// TwinCAT 3 PLC project TimeLogger_Plc
// ProgramVersion: 3.1.4023.0
// libraries:
//   Tc2_Standard, * (Beckhoff Automation GmbH)
//   Tc2_System, * (Beckhoff Automation GmbH)
//   Tc2_Utilities, * (Beckhoff Automation GmbH)
//   Tc3_Module, * (Beckhoff Automation GmbH)
// project tree:
//   DUTs/ E_EventType.TcDUT, ST_Event.TcDUT
//   / PlcTask.TcTTO
//   POUs/ EventLogger.TcPOU, FB_CsvPersistentEventStorage.TcPOU, I_PersistentEventStorage.TcIO, MAIN.TcPOU, UpdateEventTimestampWithSystemTime.TcPOU

CONFIGURATION TimeLogger_Plc
    RESOURCE PLC ON TwinCAT3
        TASK PlcTask(INTERVAL := T#10ms, PRIORITY := 20);
        PROGRAM MAIN WITH PlcTask : MAIN;
    END_RESOURCE
END_CONFIGURATION

// ---- DUTs/E_EventType.TcDUT
{attribute 'qualified_only'}
{attribute 'strict'}
{attribute 'to_string'}
TYPE E_EventType :
(
	Alarm := 0,
	Message := 1
);
END_TYPE

// ---- DUTs/ST_Event.TcDUT
TYPE ST_Event :
STRUCT
	eEventType : E_EventType; //user defined ENUM
	eEventSeverity : TcEventSeverity; // library ENUM
	nEventIdentity : UDINT;
	sEvenText : STRING(255);
	dtTimestamp : DATE_AND_TIME;
END_STRUCT
END_TYPE

// ---- POUs/I_PersistentEventStorage.TcIO
INTERFACE I_PersistentEventStorage

METHOD StoreEvent
VAR_INPUT
	stEvent : ST_Event;
END_VAR
END_METHOD

END_INTERFACE

// ---- POUs/MAIN.TcPOU
PROGRAM MAIN
VAR
	// Boolean to execute the Eventlogger in one PLC cycle
	bBoolean : BOOL := FALSE; 
	
	// Define sample values to the variables needed to add an Event
	eEventType1 : E_EventType := E_EventType.Alarm; //user defined ENUM
	eEventSeverity1 : TcEventSeverity := TcEventSeverity.Error; // library ENUM
	nEventIdentity1 : UDINT := 42;
	sEvenText1 : STRING(255) := 'This is a sample event';
	
	// Create an instance of the FB that defines the format for Persistent Event Storage
	CsvPersistentEventStorage1 : FB_CsvPersistentEventStorage;
	
	// Create one instance of our FB EventLogger, and provide interface parameter for FB_init
	EventLogger1 : EventLogger(CsvPersistentEventStorage1); 
	
END_VAR

IF bBoolean THEN
	// Add an event (in one cycle of the PLC)
	EventLogger1.AddEvent(eEventType1, eEventSeverity1, nEventIdentity1, sEvenText1); 
	bBoolean := FALSE;
END_IF

// call instance every cycle
CsvPersistentEventStorage1();

END_PROGRAM

// ---- POUs/FB_CsvPersistentEventStorage.TcPOU
FUNCTION_BLOCK FB_CsvPersistentEventStorage IMPLEMENTS I_PersistentEventStorage
VAR_INPUT
END_VAR
VAR_OUTPUT
END_VAR

VAR
	// Instantiate FB to create/open file for editing
	fbFileOpen : FB_FileOpen := (sPathName := 'C:\Events.log' , nMode := FOPEN_MODEAPPEND OR FOPEN_MODETEXT);
	
	// Instantiate FB to write into a file
	fbFilePuts : FB_FilePuts;
	
	
	// Instantiate FB to close the file
	fbFileClose : FB_FileClose;
	
	
	// create local ENUM for our State Machine
	eWriteState : (FILE_OPEN_TRIGGER, FILE_OPEN,
				                 WAIT_FOR_EVENT, 
			   WRITE_EVENT_TRIGGER, WRITE_EVENT, 
				 FILE_CLOSE_TRIGGER, FILE_CLOSE,
										 ERROR); 
	// Event to Write
	stEventWrittenToFile : ST_Event;
	
	// Variable to store the STRING to write into the file
	CsvString : T_MaxString; 	
	
END_VAR

CASE eWriteState OF
	FILE_OPEN_TRIGGER : 
		// send rising edge to request Windows to Open the File
		fbFileOpen(bExecute := TRUE);
		eWriteState := FILE_OPEN; // next step
	
	FILE_OPEN : 
		fbFileOpen(bExecute := FALSE);
		
		// Error Detection from FB OUTPUT
		IF fbFileOpen.bError THEN
			eWriteState := ERROR;
			
		// Check if we are ready to Open with Busy Flag and File Handle
		ELSIF NOT fbFileOpen.bBusy AND fbFileOpen.hFile <> 0 THEN
			eWriteState := WAIT_FOR_EVENT; // next step
			
		END_IF
	
	WAIT_FOR_EVENT :
		// Do nothing, we are waiting for the user to call us
	
	WRITE_EVENT_TRIGGER : 
		// Convert ST_Event into a CSV String (use method)
		CsvString := CreateCsvString(stEvent := stEventWrittenToFile);
		
		// send rising edge to request Windows to Write into the File
		// then send CSV String and pass the File Handle
		fbFilePuts(bExecute := TRUE,
					sLine := CsvString, 
					hFile := fbFileOpen.hFile);	
		
		eWriteState := WRITE_EVENT; // next step
	
	WRITE_EVENT : 
		fbFilePuts(bExecute := FALSE);
		
		// Error Detection from FB OUTPUT
		IF fbFilePuts.bError THEN
			eWriteState := ERROR;
		
		// Check if we are ready to write with Busy Flag 
		ELSIF NOT fbFilePuts.bBusy THEN
			eWriteState := FILE_CLOSE_TRIGGER; // next step
		END_IF
	
	FILE_CLOSE_TRIGGER : 
		// send rising edge to request Windows to Close the File
		// then pass the File Handle
		fbFileClose(bExecute := TRUE,
					hFile := fbFileOpen.hFile);	
		
		eWriteState := FILE_CLOSE; // next step
	
	FILE_CLOSE : 
		fbFileClose(bExecute := FALSE);
		
		// Error Detection from FB OUTPUT
		IF fbFileClose.bError THEN
			eWriteState := ERROR;
		
		// Check if we are ready to close with Busy Flag 
		ELSIF NOT fbFileClose.bBusy THEN
			eWriteState := FILE_OPEN_TRIGGER; // restart state machine
			
		END_IF
	
	ERROR :
		// Do nothing (for now)
		
END_CASE

METHOD PRIVATE CreateCsvString : T_MaxString
VAR_INPUT
	stEvent : REFERENCE TO ST_Event;	
END_VAR

VAR
	TempString : T_MaxString; 
	
END_VAR
TempString := TO_STRING(stEvent.eEventType);
TempString := CONCAT(STR1 := TempString, STR2 := ',');
TempString := CONCAT(STR1 := TempString, STR2 := TO_STRING(stEvent.eEventSeverity));
TempString := CONCAT(STR1 := TempString, STR2 := ',');
TempString := CONCAT(STR1 := TempString, STR2 := TO_STRING(stEvent.nEventIdentity));
TempString := CONCAT(STR1 := TempString, STR2 := ',');
TempString := CONCAT(STR1 := TempString, STR2 := stEvent.sEvenText);
TempString := CONCAT(STR1 := TempString, STR2 := ',');
TempString := CONCAT(STR1 := TempString, STR2 := TO_STRING(stEvent.dtTimestamp));
TempString := CONCAT(STR1 := TempString, STR2 := '$n');

CreateCsvString := TempString;
END_METHOD

METHOD StoreEvent
VAR_INPUT
	stEvent	: ST_Event;
END_VAR
// Here is where the CSV-writing will be done

// Are we ready to Write? 
IF eWriteState = WAIT_FOR_EVENT THEN
	// Go to next step
	eWriteState := WRITE_EVENT_TRIGGER;
	// Take Event to Write from Input
	stEventWrittenToFile := stEvent;
END_IF
END_METHOD

END_FUNCTION_BLOCK

// ---- POUs/EventLogger.TcPOU
FUNCTION_BLOCK EventLogger
VAR_INPUT
	// inputs to the function block. 
	// These are read-only, meaning you cannot modify their values within the block.
END_VAR


VAR_OUTPUT
	// outputs from the function block. 
	// The function block can modify the values of these 
END_VAR


VAR
	// local to the function block and to its methods
	// internal (instance) variables
	
	aEventBuffer : ARRAY[1..MAXIMUM_SIZE_OF_EVENT_BUFFER] OF ST_Event;
	nCurrentEventBufferIndex : INT := 0;
	
	//Create local reference of our Interface
	// FB_EventLogger USES I_PersistentEventStorage
	_PersistentEventStorage : I_PersistentEventStorage;
	
END_VAR

VAR CONSTANT
	// local to the function block and to its methods
	// these variables cannot be changed during program execution.
	
	MAXIMUM_SIZE_OF_EVENT_BUFFER : INT := 100;
	
END_VAR

(* Returns TRUE if add was succesful and FALSE if buffer is full *)
METHOD PUBLIC AddEvent : BOOL
VAR_INPUT
	// user input
	eEventType : E_EventType; //user defined ENUM
	eEventSeverity : TcEventSeverity; // library ENUM
	nEventIdentity : UDINT;
	sEvenText : STRING(255);
	
END_VAR
//Check if the event buffer is full using a private method
IF NOT IsEventBufferFull () THEN
	
	nCurrentEventBufferIndex := nCurrentEventBufferIndex + 1;
	
	// from user input, fill buffer
	aEventBuffer[nCurrentEventBufferIndex].eEventType := eEventType;
	aEventBuffer[nCurrentEventBufferIndex].eEventSeverity := eEventSeverity;
	aEventBuffer[nCurrentEventBufferIndex].nEventIdentity := nEventIdentity;
	aEventBuffer[nCurrentEventBufferIndex].sEvenText := sEvenText;
	
	// using our function, fill the date and time stamp
	// input current event to the function
	// updates only date and type stamp of the input event
	UpdateEventTimestampWithSystemTime(stEvent := aEventBuffer[nCurrentEventBufferIndex]);
	
	AddEvent := TRUE; // add was succesful
ELSE
	AddEvent := FALSE; // buffer is full
END_IF

// Here we want to store the event persistently
_PersistentEventStorage.StoreEvent(stEvent := aEventBuffer[nCurrentEventBufferIndex]);
END_METHOD

METHOD FB_init : BOOL
VAR_INPUT
	bInitRetains : BOOL; // if TRUE, the retain variables are initialized (warm start / cold start)
	bInCopyCode : BOOL;  // if TRUE, the instance afterwards gets moved into the copy code (online change)
	
	// Making a reference to the Interface I_PersistentEventStorage
	// This Interface is for Storing Events Persistently	
	iPersistentEventStorage : I_PersistentEventStorage; 
END_VAR
// store reference locally in the FB when FB_init method executes
// this allows all methods in the FB to have access to it
_PersistentEventStorage := iPersistentEventStorage;
END_METHOD

METHOD PRIVATE IsEventBufferFull : BOOL
//Check if the event buffer is full
IF (nCurrentEventBufferIndex + 1) > MAXIMUM_SIZE_OF_EVENT_BUFFER THEN
	IsEventBufferFull := TRUE; //method returns TRUE, it is full
ELSE 
	IsEventBufferFull := FALSE; //method returns FALSE, it is not full
END_IF
END_METHOD

END_FUNCTION_BLOCK

// ---- POUs/UpdateEventTimestampWithSystemTime.TcPOU
FUNCTION UpdateEventTimestampWithSystemTime
VAR_INPUT
	stEvent : REFERENCE TO ST_Event;
END_VAR
VAR
	fbGETSYSTEMTIME : GETSYSTEMTIME;
	stFileTime : T_FILETIME; // requires Tc2_Utilities
END_VAR

// The function block writes on stFileTime (VAR_OUTPUT) in T_FILETIME format 
fbGETSYSTEMTIME(timeLoDW => stFileTime.dwLowDateTime,
				timeHiDW => stFileTime.dwHighDateTime);

// Overwrites the Timestamp of stEvent using the FILETIME_TO_DT function
stEvent.dtTimestamp := FILETIME_TO_DT(fileTime := stFileTime);

END_FUNCTION
